PROGRAM P_AxisControl
VAR
END_VAR

//Axis Control program based on youtube series Twincat 3 NC Videos MB05a until MB17b plus MB22 by @electricalautomation https://www.youtube.com/watch?v=BxRAOdTks9I&list=PL762SfoJC-e8NbAUQ-H7a_TOdqrlBPCw4&index=25

IF G_Inputs.bManualModeSelector THEN
	Manual_mode();
ELSIF G_Inputs.bAutoModeSelector THEN
	Auto_mode();
ELSE
	GVL_AXIS1.lrBC_PowerOverride := 0;
	GVL_AXIS1.bBC_StopExe := TRUE;
	GVL_AXIS2.lrSJ_PowerOverride := 0;
	GVL_AXIS2.bSJ_StopExe := TRUE;
	GVL_AXIS3.lrTC_PowerOverride := 0;
	GVL_AXIS3.bTC_StopExe := TRUE;
	GVL_AXIS4.lrWM_PowerOverride := 0;
	GVL_AXIS4.bWM_StopExe := TRUE;
END_IF

METHOD Auto_mode : BOOL
VAR_INPUT
END_VAR
//AXIS 1 Main arm actuator

GVL_AXIS1.lrBC_PowerOverride := 100;

GVL_AXIS1.bBC_ResetExe := G_Inputs.bJoystickLeftEnable OR G_Inputs.bGreenButton OR GVL_AXIS1.bBC_MoveAbsDone;

//Power Enable
GVL_AXIS1.bBC_PowerEnCmd := G_Inputs.bAutoModeSelector;
GVL_AXIS1.bBC_PowerEnNegative := G_Inputs.bAutoModeSelector;
GVL_AXIS1.bBC_PowerEnPositive := G_Inputs.bAutoModeSelector;

GVL_AXIS1.lrBC_MoveAbsPosition := GVL_InverseKinematics.fStrokeActuatorMainInverse*1000;
GVL_AXIS1.lrBC_MoveAbsVelocity := 30;
GVL_AXIS1.bBC_MoveAbsExe := G_Inputs.bGreenButton;


//Position control
IF G_Inputs.bJoystickLeftEnable AND GVL_AXIS1.bBC_MoveAbsDone THEN
	GVL_AXIS1.bBC_ExtSetGenDisExe := FALSE;
	GVL_AXIS1.bBC_ExtSetGenEnaExe := TRUE;
ELSE
	GVL_AXIS1.bBC_ExtSetGenDisExe := TRUE;
	GVL_AXIS1.bBC_ExtSetGenEnaExe := FALSE;
END_IF


GVL_AXIS1.lrBC_MoveAddPos := GVL_InverseKinematics.fStrokeActuatorMainInverse*1000;


//Update axis
AXIS1_LD_Auto();


//Axis 3 Knuckle arm actuator

GVL_AXIS3.lrTC_PowerOverride := 100;

GVL_AXIS3.bTC_ResetExe := G_Inputs.bJoystickLeftEnable OR G_Inputs.bGreenButton OR GVL_AXIS3.bTC_MoveAbsDone;

//Power Enable
GVL_AXIS3.bTC_PowerEnCmd := G_Inputs.bAutoModeSelector;
GVL_AXIS3.bTC_PowerEnNegative := G_Inputs.bAutoModeSelector;
GVL_AXIS3.bTC_PowerEnPositive := G_Inputs.bAutoModeSelector;

GVL_AXIS3.lrTC_MoveAbsPosition := GVL_InverseKinematics.fStrokeActuatorKnuckleInverse*1000;
GVL_AXIS3.lrTC_MoveAbsVelocity := 30;
GVL_AXIS3.bTC_MoveAbsExe := G_Inputs.bGreenButton;


//Position control
IF G_Inputs.bJoystickLeftEnable AND GVL_AXIS3.bTC_MoveAbsDone THEN
	GVL_AXIS3.bTC_ExtSetGenDisExe := FALSE;
	GVL_AXIS3.bTC_ExtSetGenEnaExe := TRUE;
ELSE
	GVL_AXIS3.bTC_ExtSetGenDisExe := TRUE;
	GVL_AXIS3.bTC_ExtSetGenEnaExe := FALSE;
END_IF


GVL_AXIS3.lrTC_MoveAddPos := GVL_InverseKinematics.fStrokeActuatorKnuckleInverse*1000;


//Update axis
AXIS3_LD_Auto();


//Axis 4 Winch motor

GVL_AXIS4.lrWM_PowerOverride := 100;

GVL_AXIS4.bWM_ResetExe := G_Inputs.bJoystickRightEnable OR G_Inputs.bGreenButton OR GVL_AXIS1.bBC_MoveAbsDone;

//Power Enable
GVL_AXIS4.bWM_PowerEnCmd := G_Inputs.bAutoModeSelector;
GVL_AXIS4.bWM_PowerEnNegative := G_Inputs.bAutoModeSelector;
GVL_AXIS4.bWM_PowerEnPositive := G_Inputs.bAutoModeSelector;


GVL_AXIS4.lrWM_MoveAbsPosition := G_MachineControl.fWinchMotorAngleRef;
GVL_AXIS4.lrWM_MoveAbsVelocity := 10;
GVL_AXIS4.bWM_MoveAbsExe := G_Inputs.bGreenButton;


//Position control
IF G_Inputs.bJoystickRightEnable AND GVL_AXIS4.bWM_MoveAbsDone  THEN
	GVL_AXIS4.bWM_ExtSetGenDisExe := FALSE;
	GVL_AXIS4.bWM_ExtSetGenEnaExe := TRUE;
ELSE
	GVL_AXIS4.bWM_ExtSetGenDisExe := TRUE;
	GVL_AXIS4.bWM_ExtSetGenEnaExe := FALSE;
END_IF

(*
//Position control
IF G_Inputs.bJoystickRightEnable THEN
	GVL_AXIS4.bWM_ExtSetGenDisExe := FALSE;
	GVL_AXIS4.bWM_ExtSetGenEnaExe := TRUE;
ELSE
	GVL_AXIS4.bWM_ExtSetGenDisExe := TRUE;
	GVL_AXIS4.bWM_ExtSetGenEnaExe := FALSE;
END_IF
*)

GVL_AXIS4.lrWM_MoveAddPos := G_MachineControl.fPosRefWinch*180/PI; //Convert to degrees


//Update axis
AXIS4_LD_Auto();
END_METHOD

METHOD AXIS1_LD : BOOL
VAR_INPUT
END_VAR
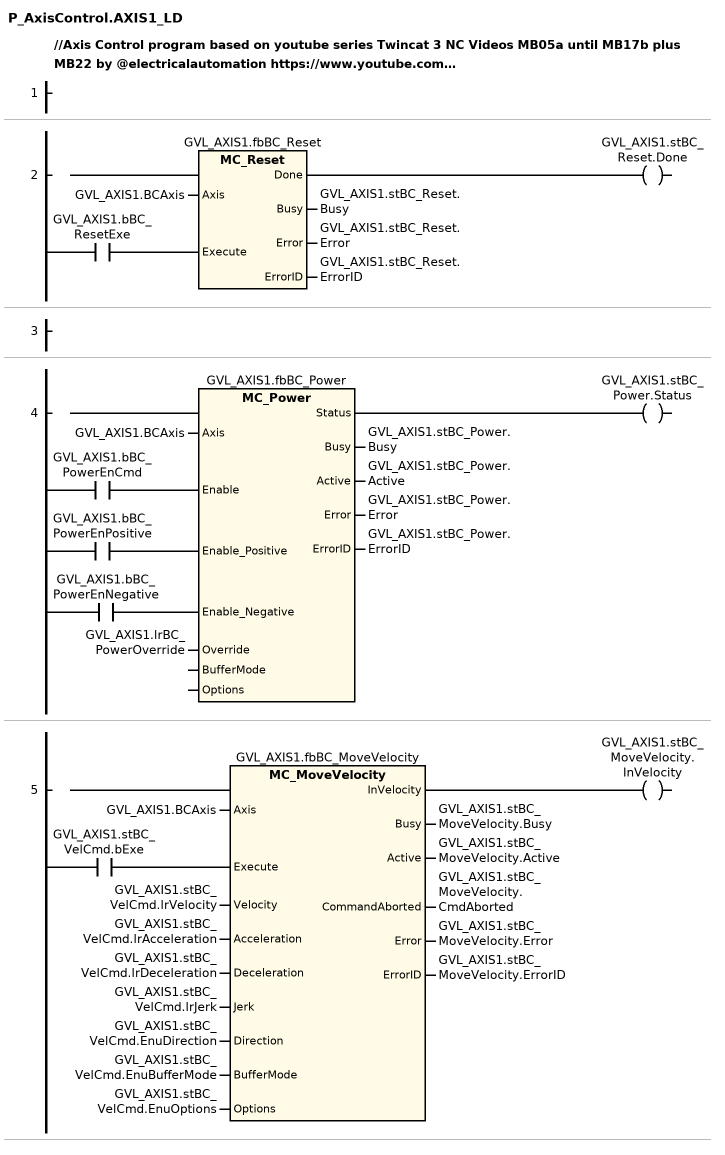
// NETWORK 1: //Axis Control program based on youtube series Twincat 3 NC Videos MB05a until MB17b plus MB22 by @electricalautomation https://www.youtube.com/watch?v=BxRAOdTks9I&list=PL762SfoJC-e8NbAUQ-H7a_TOdqrlBPCw4&index=25

// NETWORK 2
GVL_AXIS1.fbBC_Reset(
    Axis := GVL_AXIS1.BCAxis,
    Execute := GVL_AXIS1.bBC_ResetExe,
    Busy => GVL_AXIS1.stBC_Reset.Busy,
    Error => GVL_AXIS1.stBC_Reset.Error,
    ErrorID => GVL_AXIS1.stBC_Reset.ErrorID); // MC_Reset
GVL_AXIS1.stBC_Reset.Done := GVL_AXIS1.fbBC_Reset.Done;

// NETWORK 3

// NETWORK 4
GVL_AXIS1.fbBC_Power(
    Axis := GVL_AXIS1.BCAxis,
    Enable := GVL_AXIS1.bBC_PowerEnCmd,
    Enable_Positive := GVL_AXIS1.bBC_PowerEnPositive,
    Enable_Negative := GVL_AXIS1.bBC_PowerEnNegative,
    Override := GVL_AXIS1.lrBC_PowerOverride,
    Busy => GVL_AXIS1.stBC_Power.Busy,
    Active => GVL_AXIS1.stBC_Power.Active,
    Error => GVL_AXIS1.stBC_Power.Error,
    ErrorID => GVL_AXIS1.stBC_Power.ErrorID); // MC_Power
GVL_AXIS1.stBC_Power.Status := GVL_AXIS1.fbBC_Power.Status;

// NETWORK 5
GVL_AXIS1.fbBC_MoveVelocity(
    Axis := GVL_AXIS1.BCAxis,
    Execute := GVL_AXIS1.stBC_VelCmd.bExe,
    Velocity := GVL_AXIS1.stBC_VelCmd.lrVelocity,
    Acceleration := GVL_AXIS1.stBC_VelCmd.lrAcceleration,
    Deceleration := GVL_AXIS1.stBC_VelCmd.lrDeceleration,
    Jerk := GVL_AXIS1.stBC_VelCmd.lrJerk,
    Direction := GVL_AXIS1.stBC_VelCmd.EnuDirection,
    BufferMode := GVL_AXIS1.stBC_VelCmd.EnuBufferMode,
    Options := GVL_AXIS1.stBC_VelCmd.EnuOptions,
    Busy => GVL_AXIS1.stBC_MoveVelocity.Busy,
    Active => GVL_AXIS1.stBC_MoveVelocity.Active,
    CommandAborted => GVL_AXIS1.stBC_MoveVelocity.CmdAborted,
    Error => GVL_AXIS1.stBC_MoveVelocity.Error,
    ErrorID => GVL_AXIS1.stBC_MoveVelocity.ErrorID); // MC_MoveVelocity
GVL_AXIS1.stBC_MoveVelocity.InVelocity := GVL_AXIS1.fbBC_MoveVelocity.InVelocity;
END_METHOD

METHOD AXIS1_LD_Auto : BOOL
VAR_INPUT
END_VAR
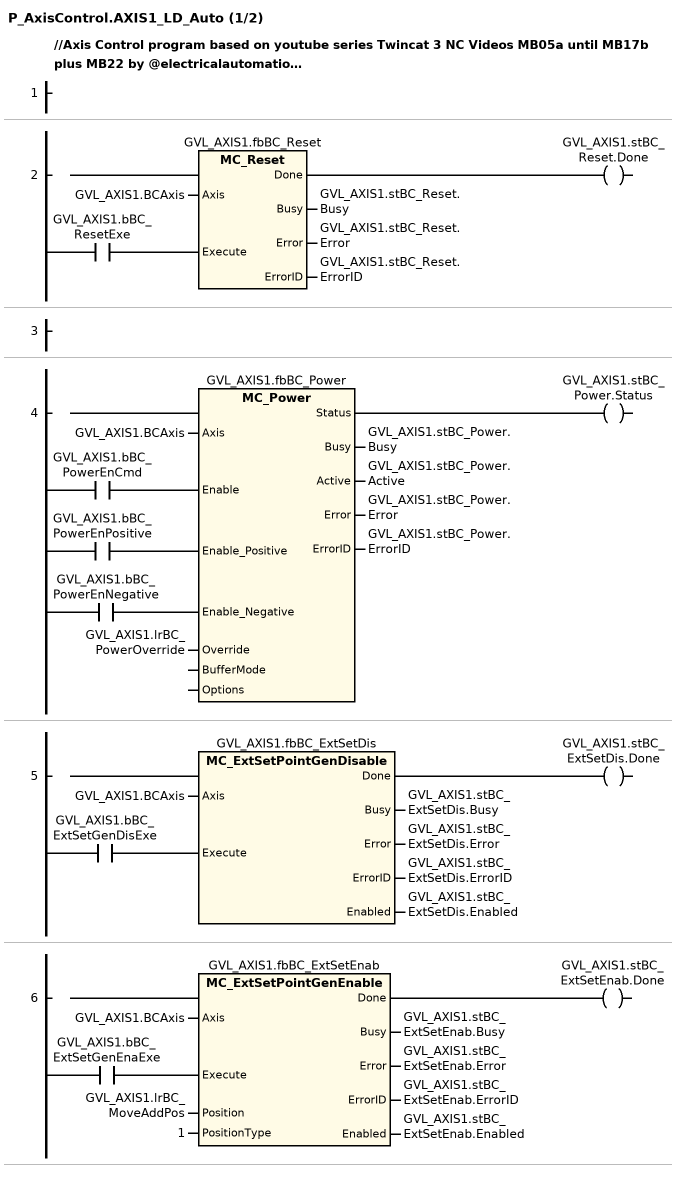
// NETWORK 1: //Axis Control program based on youtube series Twincat 3 NC Videos MB05a until MB17b plus MB22 by @electricalautomation https://www.youtube.com/watch?v=BxRAOdTks9I&list=PL762SfoJC-e8NbAUQ-H7a_TOdqrlBPCw4&index=25

// NETWORK 2
GVL_AXIS1.fbBC_Reset(
    Axis := GVL_AXIS1.BCAxis,
    Execute := GVL_AXIS1.bBC_ResetExe,
    Busy => GVL_AXIS1.stBC_Reset.Busy,
    Error => GVL_AXIS1.stBC_Reset.Error,
    ErrorID => GVL_AXIS1.stBC_Reset.ErrorID); // MC_Reset
GVL_AXIS1.stBC_Reset.Done := GVL_AXIS1.fbBC_Reset.Done;

// NETWORK 3

// NETWORK 4
GVL_AXIS1.fbBC_Power(
    Axis := GVL_AXIS1.BCAxis,
    Enable := GVL_AXIS1.bBC_PowerEnCmd,
    Enable_Positive := GVL_AXIS1.bBC_PowerEnPositive,
    Enable_Negative := GVL_AXIS1.bBC_PowerEnNegative,
    Override := GVL_AXIS1.lrBC_PowerOverride,
    Busy => GVL_AXIS1.stBC_Power.Busy,
    Active => GVL_AXIS1.stBC_Power.Active,
    Error => GVL_AXIS1.stBC_Power.Error,
    ErrorID => GVL_AXIS1.stBC_Power.ErrorID); // MC_Power
GVL_AXIS1.stBC_Power.Status := GVL_AXIS1.fbBC_Power.Status;

// NETWORK 5
GVL_AXIS1.fbBC_ExtSetDis(
    Axis := GVL_AXIS1.BCAxis,
    Execute := GVL_AXIS1.bBC_ExtSetGenDisExe,
    Busy => GVL_AXIS1.stBC_ExtSetDis.Busy,
    Error => GVL_AXIS1.stBC_ExtSetDis.Error,
    ErrorID => GVL_AXIS1.stBC_ExtSetDis.ErrorID,
    Enabled => GVL_AXIS1.stBC_ExtSetDis.Enabled); // MC_ExtSetPointGenDisable
GVL_AXIS1.stBC_ExtSetDis.Done := GVL_AXIS1.fbBC_ExtSetDis.Done;

// NETWORK 6
GVL_AXIS1.fbBC_ExtSetEnab(
    Axis := GVL_AXIS1.BCAxis,
    Execute := GVL_AXIS1.bBC_ExtSetGenEnaExe,
    Position := GVL_AXIS1.lrBC_MoveAddPos,
    PositionType := 1,
    Busy => GVL_AXIS1.stBC_ExtSetEnab.Busy,
    Error => GVL_AXIS1.stBC_ExtSetEnab.Error,
    ErrorID => GVL_AXIS1.stBC_ExtSetEnab.ErrorID,
    Enabled => GVL_AXIS1.stBC_ExtSetEnab.Enabled); // MC_ExtSetPointGenEnable
GVL_AXIS1.stBC_ExtSetEnab.Done := GVL_AXIS1.fbBC_ExtSetEnab.Done;

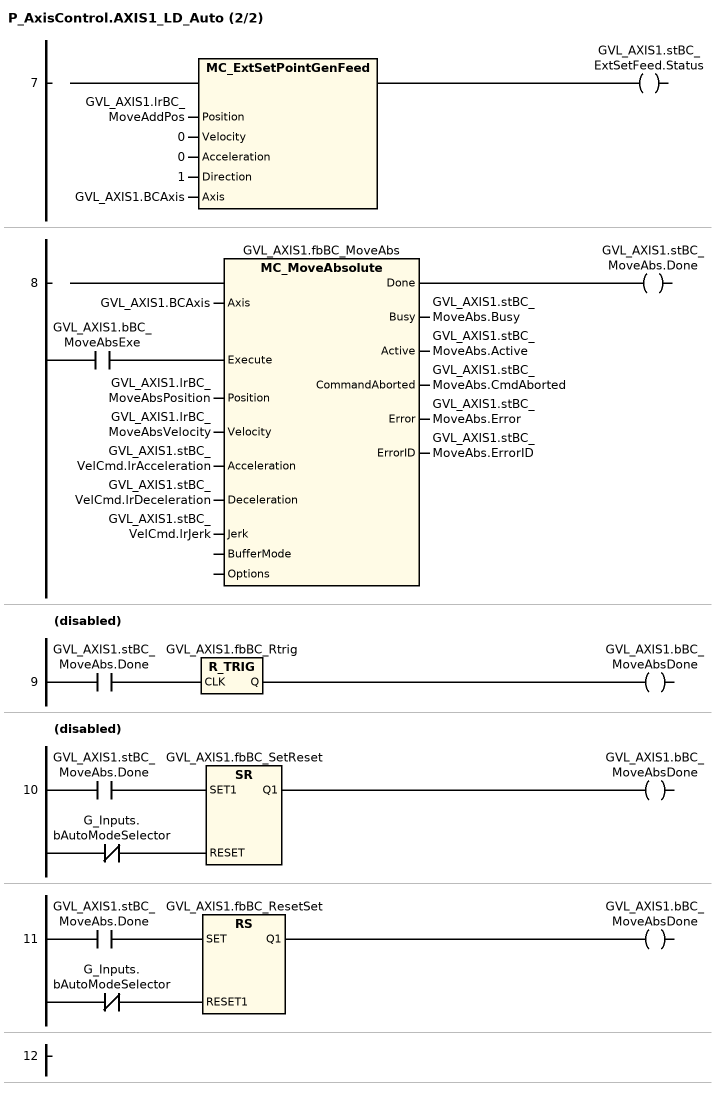
// NETWORK 7
GVL_AXIS1.stBC_ExtSetFeed.Status := MC_ExtSetPointGenFeed(Position := GVL_AXIS1.lrBC_MoveAddPos, Velocity := 0, Acceleration := 0, Direction := 1, Axis := GVL_AXIS1.BCAxis);

// NETWORK 8
GVL_AXIS1.fbBC_MoveAbs(
    Axis := GVL_AXIS1.BCAxis,
    Execute := GVL_AXIS1.bBC_MoveAbsExe,
    Position := GVL_AXIS1.lrBC_MoveAbsPosition,
    Velocity := GVL_AXIS1.lrBC_MoveAbsVelocity,
    Acceleration := GVL_AXIS1.stBC_VelCmd.lrAcceleration,
    Deceleration := GVL_AXIS1.stBC_VelCmd.lrDeceleration,
    Jerk := GVL_AXIS1.stBC_VelCmd.lrJerk,
    Busy => GVL_AXIS1.stBC_MoveAbs.Busy,
    Active => GVL_AXIS1.stBC_MoveAbs.Active,
    CommandAborted => GVL_AXIS1.stBC_MoveAbs.CmdAborted,
    Error => GVL_AXIS1.stBC_MoveAbs.Error,
    ErrorID => GVL_AXIS1.stBC_MoveAbs.ErrorID); // MC_MoveAbsolute
GVL_AXIS1.stBC_MoveAbs.Done := GVL_AXIS1.fbBC_MoveAbs.Done;

// NETWORK 9 (disabled)
// GVL_AXIS1.fbBC_Rtrig(CLK := GVL_AXIS1.stBC_MoveAbs.Done); // R_TRIG
// GVL_AXIS1.bBC_MoveAbsDone := GVL_AXIS1.fbBC_Rtrig.Q;

// NETWORK 10 (disabled)
// GVL_AXIS1.fbBC_SetReset(SET1 := GVL_AXIS1.stBC_MoveAbs.Done, RESET := NOT G_Inputs.bAutoModeSelector); // SR
// GVL_AXIS1.bBC_MoveAbsDone := GVL_AXIS1.fbBC_SetReset.Q1;

// NETWORK 11
GVL_AXIS1.fbBC_ResetSet(SET := GVL_AXIS1.stBC_MoveAbs.Done, RESET1 := NOT G_Inputs.bAutoModeSelector); // RS
GVL_AXIS1.bBC_MoveAbsDone := GVL_AXIS1.fbBC_ResetSet.Q1;

// NETWORK 12
END_METHOD

METHOD AXIS2_LD : BOOL
VAR_INPUT
END_VAR
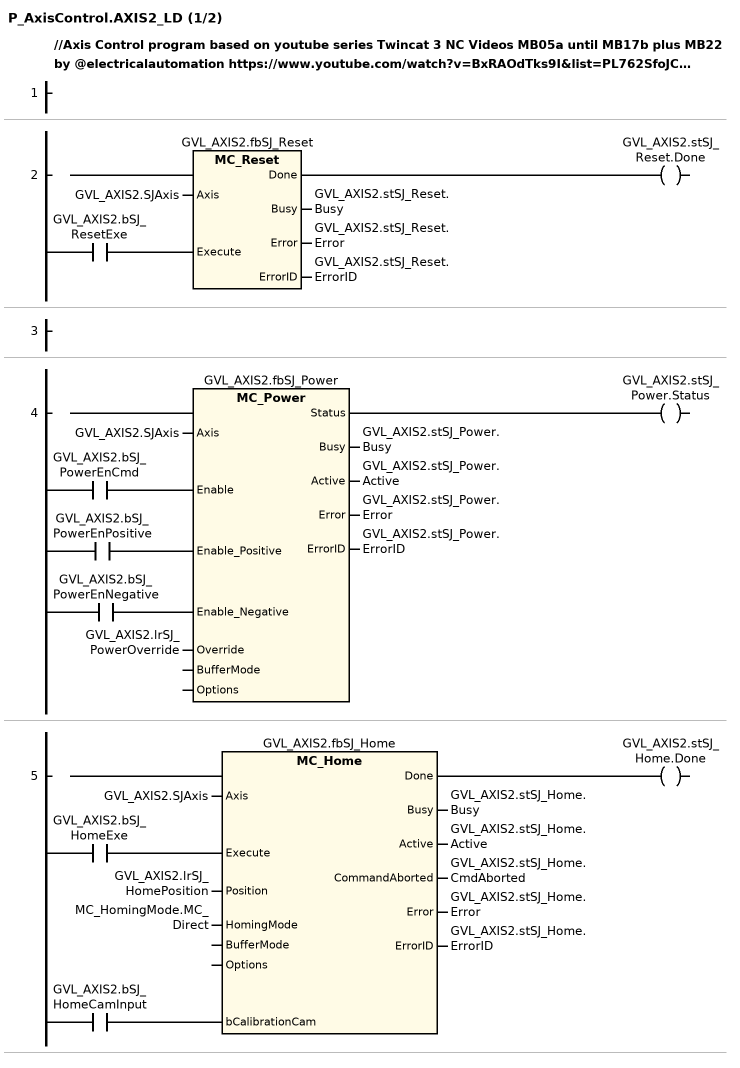
// NETWORK 1: //Axis Control program based on youtube series Twincat 3 NC Videos MB05a until MB17b plus MB22 by @electricalautomation https://www.youtube.com/watch?v=BxRAOdTks9I&list=PL762SfoJC-e8NbAUQ-H7a_TOdqrlBPCw4&index=25

// NETWORK 2
GVL_AXIS2.fbSJ_Reset(
    Axis := GVL_AXIS2.SJAxis,
    Execute := GVL_AXIS2.bSJ_ResetExe,
    Busy => GVL_AXIS2.stSJ_Reset.Busy,
    Error => GVL_AXIS2.stSJ_Reset.Error,
    ErrorID => GVL_AXIS2.stSJ_Reset.ErrorID); // MC_Reset
GVL_AXIS2.stSJ_Reset.Done := GVL_AXIS2.fbSJ_Reset.Done;

// NETWORK 3

// NETWORK 4
GVL_AXIS2.fbSJ_Power(
    Axis := GVL_AXIS2.SJAxis,
    Enable := GVL_AXIS2.bSJ_PowerEnCmd,
    Enable_Positive := GVL_AXIS2.bSJ_PowerEnPositive,
    Enable_Negative := GVL_AXIS2.bSJ_PowerEnNegative,
    Override := GVL_AXIS2.lrSJ_PowerOverride,
    Busy => GVL_AXIS2.stSJ_Power.Busy,
    Active => GVL_AXIS2.stSJ_Power.Active,
    Error => GVL_AXIS2.stSJ_Power.Error,
    ErrorID => GVL_AXIS2.stSJ_Power.ErrorID); // MC_Power
GVL_AXIS2.stSJ_Power.Status := GVL_AXIS2.fbSJ_Power.Status;

// NETWORK 5
GVL_AXIS2.fbSJ_Home(
    Axis := GVL_AXIS2.SJAxis,
    Execute := GVL_AXIS2.bSJ_HomeExe,
    Position := GVL_AXIS2.lrSJ_HomePosition,
    HomingMode := MC_HomingMode.MC_Direct,
    bCalibrationCam := GVL_AXIS2.bSJ_HomeCamInput,
    Busy => GVL_AXIS2.stSJ_Home.Busy,
    Active => GVL_AXIS2.stSJ_Home.Active,
    CommandAborted => GVL_AXIS2.stSJ_Home.CmdAborted,
    Error => GVL_AXIS2.stSJ_Home.Error,
    ErrorID => GVL_AXIS2.stSJ_Home.ErrorID); // MC_Home
GVL_AXIS2.stSJ_Home.Done := GVL_AXIS2.fbSJ_Home.Done;

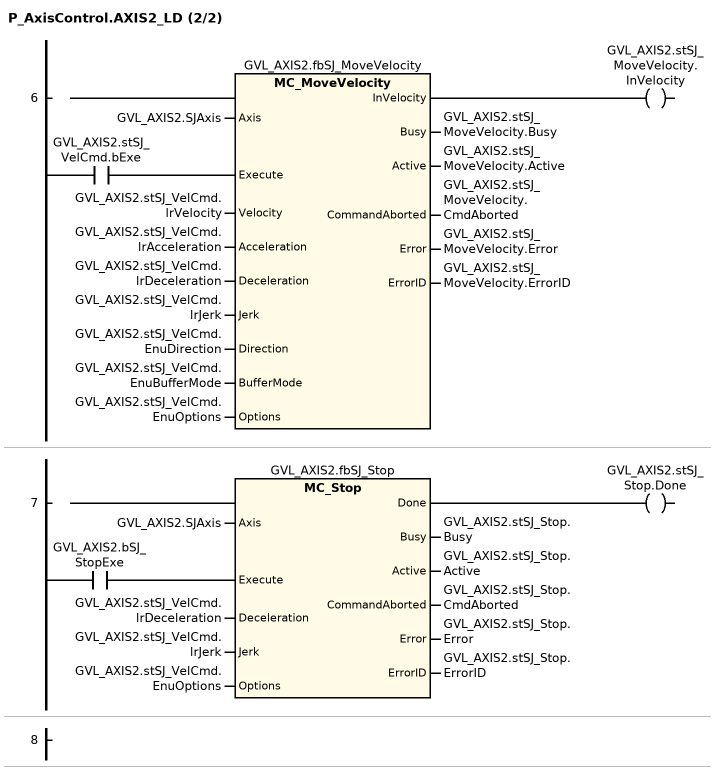
// NETWORK 6
GVL_AXIS2.fbSJ_MoveVelocity(
    Axis := GVL_AXIS2.SJAxis,
    Execute := GVL_AXIS2.stSJ_VelCmd.bExe,
    Velocity := GVL_AXIS2.stSJ_VelCmd.lrVelocity,
    Acceleration := GVL_AXIS2.stSJ_VelCmd.lrAcceleration,
    Deceleration := GVL_AXIS2.stSJ_VelCmd.lrDeceleration,
    Jerk := GVL_AXIS2.stSJ_VelCmd.lrJerk,
    Direction := GVL_AXIS2.stSJ_VelCmd.EnuDirection,
    BufferMode := GVL_AXIS2.stSJ_VelCmd.EnuBufferMode,
    Options := GVL_AXIS2.stSJ_VelCmd.EnuOptions,
    Busy => GVL_AXIS2.stSJ_MoveVelocity.Busy,
    Active => GVL_AXIS2.stSJ_MoveVelocity.Active,
    CommandAborted => GVL_AXIS2.stSJ_MoveVelocity.CmdAborted,
    Error => GVL_AXIS2.stSJ_MoveVelocity.Error,
    ErrorID => GVL_AXIS2.stSJ_MoveVelocity.ErrorID); // MC_MoveVelocity
GVL_AXIS2.stSJ_MoveVelocity.InVelocity := GVL_AXIS2.fbSJ_MoveVelocity.InVelocity;

// NETWORK 7
GVL_AXIS2.fbSJ_Stop(
    Axis := GVL_AXIS2.SJAxis,
    Execute := GVL_AXIS2.bSJ_StopExe,
    Deceleration := GVL_AXIS2.stSJ_VelCmd.lrDeceleration,
    Jerk := GVL_AXIS2.stSJ_VelCmd.lrJerk,
    Options := GVL_AXIS2.stSJ_VelCmd.EnuOptions,
    Busy => GVL_AXIS2.stSJ_Stop.Busy,
    Active => GVL_AXIS2.stSJ_Stop.Active,
    CommandAborted => GVL_AXIS2.stSJ_Stop.CmdAborted,
    Error => GVL_AXIS2.stSJ_Stop.Error,
    ErrorID => GVL_AXIS2.stSJ_Stop.ErrorID); // MC_Stop
GVL_AXIS2.stSJ_Stop.Done := GVL_AXIS2.fbSJ_Stop.Done;

// NETWORK 8
END_METHOD

METHOD AXIS3_LD : BOOL
VAR_INPUT
END_VAR
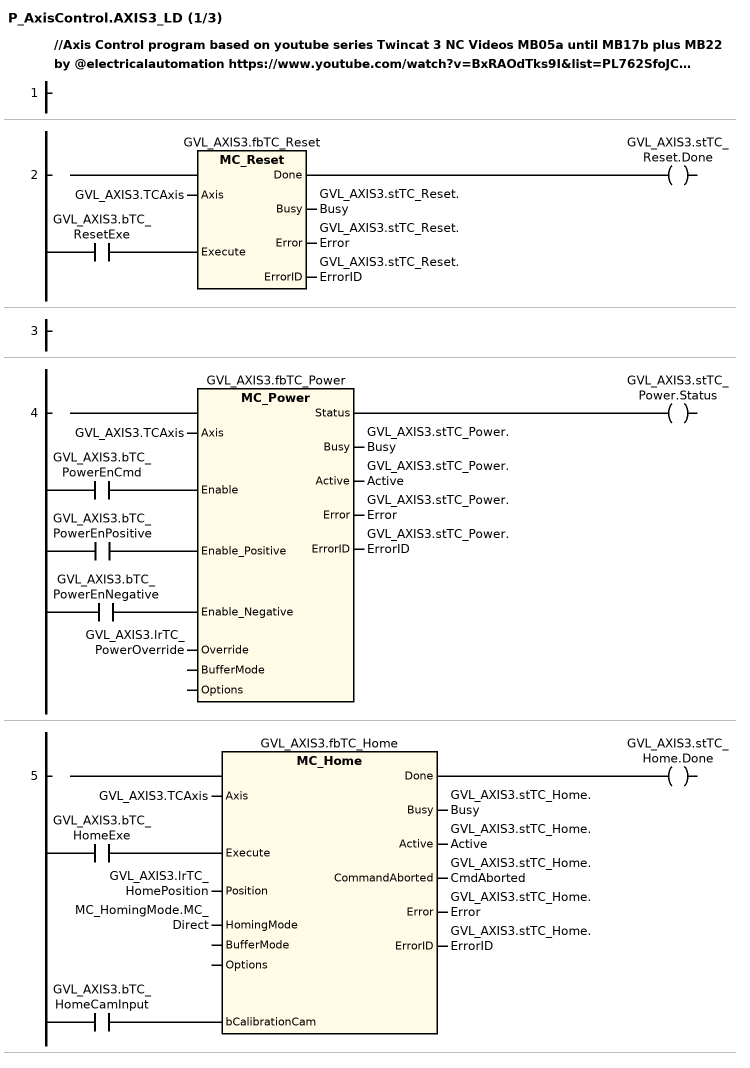
// NETWORK 1: //Axis Control program based on youtube series Twincat 3 NC Videos MB05a until MB17b plus MB22 by @electricalautomation https://www.youtube.com/watch?v=BxRAOdTks9I&list=PL762SfoJC-e8NbAUQ-H7a_TOdqrlBPCw4&index=25

// NETWORK 2
GVL_AXIS3.fbTC_Reset(
    Axis := GVL_AXIS3.TCAxis,
    Execute := GVL_AXIS3.bTC_ResetExe,
    Busy => GVL_AXIS3.stTC_Reset.Busy,
    Error => GVL_AXIS3.stTC_Reset.Error,
    ErrorID => GVL_AXIS3.stTC_Reset.ErrorID); // MC_Reset
GVL_AXIS3.stTC_Reset.Done := GVL_AXIS3.fbTC_Reset.Done;

// NETWORK 3

// NETWORK 4
GVL_AXIS3.fbTC_Power(
    Axis := GVL_AXIS3.TCAxis,
    Enable := GVL_AXIS3.bTC_PowerEnCmd,
    Enable_Positive := GVL_AXIS3.bTC_PowerEnPositive,
    Enable_Negative := GVL_AXIS3.bTC_PowerEnNegative,
    Override := GVL_AXIS3.lrTC_PowerOverride,
    Busy => GVL_AXIS3.stTC_Power.Busy,
    Active => GVL_AXIS3.stTC_Power.Active,
    Error => GVL_AXIS3.stTC_Power.Error,
    ErrorID => GVL_AXIS3.stTC_Power.ErrorID); // MC_Power
GVL_AXIS3.stTC_Power.Status := GVL_AXIS3.fbTC_Power.Status;

// NETWORK 5
GVL_AXIS3.fbTC_Home(
    Axis := GVL_AXIS3.TCAxis,
    Execute := GVL_AXIS3.bTC_HomeExe,
    Position := GVL_AXIS3.lrTC_HomePosition,
    HomingMode := MC_HomingMode.MC_Direct,
    bCalibrationCam := GVL_AXIS3.bTC_HomeCamInput,
    Busy => GVL_AXIS3.stTC_Home.Busy,
    Active => GVL_AXIS3.stTC_Home.Active,
    CommandAborted => GVL_AXIS3.stTC_Home.CmdAborted,
    Error => GVL_AXIS3.stTC_Home.Error,
    ErrorID => GVL_AXIS3.stTC_Home.ErrorID); // MC_Home
GVL_AXIS3.stTC_Home.Done := GVL_AXIS3.fbTC_Home.Done;

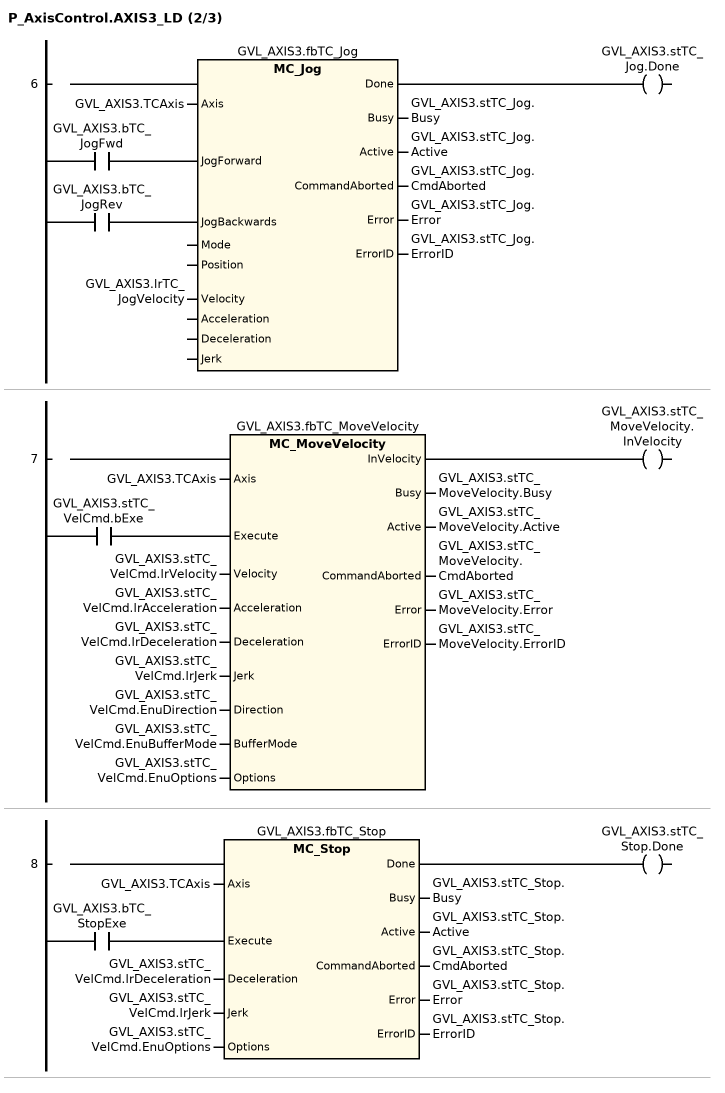
// NETWORK 6
GVL_AXIS3.fbTC_Jog(
    Axis := GVL_AXIS3.TCAxis,
    JogForward := GVL_AXIS3.bTC_JogFwd,
    JogBackwards := GVL_AXIS3.bTC_JogRev,
    Velocity := GVL_AXIS3.lrTC_JogVelocity,
    Busy => GVL_AXIS3.stTC_Jog.Busy,
    Active => GVL_AXIS3.stTC_Jog.Active,
    CommandAborted => GVL_AXIS3.stTC_Jog.CmdAborted,
    Error => GVL_AXIS3.stTC_Jog.Error,
    ErrorID => GVL_AXIS3.stTC_Jog.ErrorID); // MC_Jog
GVL_AXIS3.stTC_Jog.Done := GVL_AXIS3.fbTC_Jog.Done;

// NETWORK 7
GVL_AXIS3.fbTC_MoveVelocity(
    Axis := GVL_AXIS3.TCAxis,
    Execute := GVL_AXIS3.stTC_VelCmd.bExe,
    Velocity := GVL_AXIS3.stTC_VelCmd.lrVelocity,
    Acceleration := GVL_AXIS3.stTC_VelCmd.lrAcceleration,
    Deceleration := GVL_AXIS3.stTC_VelCmd.lrDeceleration,
    Jerk := GVL_AXIS3.stTC_VelCmd.lrJerk,
    Direction := GVL_AXIS3.stTC_VelCmd.EnuDirection,
    BufferMode := GVL_AXIS3.stTC_VelCmd.EnuBufferMode,
    Options := GVL_AXIS3.stTC_VelCmd.EnuOptions,
    Busy => GVL_AXIS3.stTC_MoveVelocity.Busy,
    Active => GVL_AXIS3.stTC_MoveVelocity.Active,
    CommandAborted => GVL_AXIS3.stTC_MoveVelocity.CmdAborted,
    Error => GVL_AXIS3.stTC_MoveVelocity.Error,
    ErrorID => GVL_AXIS3.stTC_MoveVelocity.ErrorID); // MC_MoveVelocity
GVL_AXIS3.stTC_MoveVelocity.InVelocity := GVL_AXIS3.fbTC_MoveVelocity.InVelocity;

// NETWORK 8
GVL_AXIS3.fbTC_Stop(
    Axis := GVL_AXIS3.TCAxis,
    Execute := GVL_AXIS3.bTC_StopExe,
    Deceleration := GVL_AXIS3.stTC_VelCmd.lrDeceleration,
    Jerk := GVL_AXIS3.stTC_VelCmd.lrJerk,
    Options := GVL_AXIS3.stTC_VelCmd.EnuOptions,
    Busy => GVL_AXIS3.stTC_Stop.Busy,
    Active => GVL_AXIS3.stTC_Stop.Active,
    CommandAborted => GVL_AXIS3.stTC_Stop.CmdAborted,
    Error => GVL_AXIS3.stTC_Stop.Error,
    ErrorID => GVL_AXIS3.stTC_Stop.ErrorID); // MC_Stop
GVL_AXIS3.stTC_Stop.Done := GVL_AXIS3.fbTC_Stop.Done;

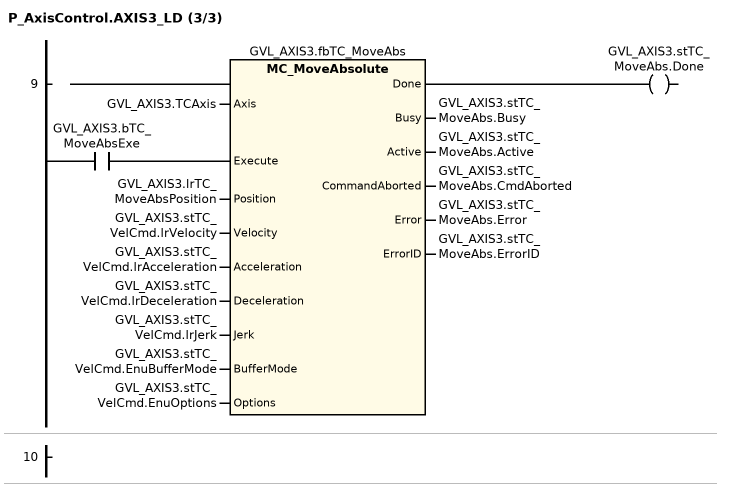
// NETWORK 9
GVL_AXIS3.fbTC_MoveAbs(
    Axis := GVL_AXIS3.TCAxis,
    Execute := GVL_AXIS3.bTC_MoveAbsExe,
    Position := GVL_AXIS3.lrTC_MoveAbsPosition,
    Velocity := GVL_AXIS3.stTC_VelCmd.lrVelocity,
    Acceleration := GVL_AXIS3.stTC_VelCmd.lrAcceleration,
    Deceleration := GVL_AXIS3.stTC_VelCmd.lrDeceleration,
    Jerk := GVL_AXIS3.stTC_VelCmd.lrJerk,
    BufferMode := GVL_AXIS3.stTC_VelCmd.EnuBufferMode,
    Options := GVL_AXIS3.stTC_VelCmd.EnuOptions,
    Busy => GVL_AXIS3.stTC_MoveAbs.Busy,
    Active => GVL_AXIS3.stTC_MoveAbs.Active,
    CommandAborted => GVL_AXIS3.stTC_MoveAbs.CmdAborted,
    Error => GVL_AXIS3.stTC_MoveAbs.Error,
    ErrorID => GVL_AXIS3.stTC_MoveAbs.ErrorID); // MC_MoveAbsolute
GVL_AXIS3.stTC_MoveAbs.Done := GVL_AXIS3.fbTC_MoveAbs.Done;

// NETWORK 10
END_METHOD

METHOD AXIS3_LD_Auto : BOOL
VAR_INPUT
END_VAR
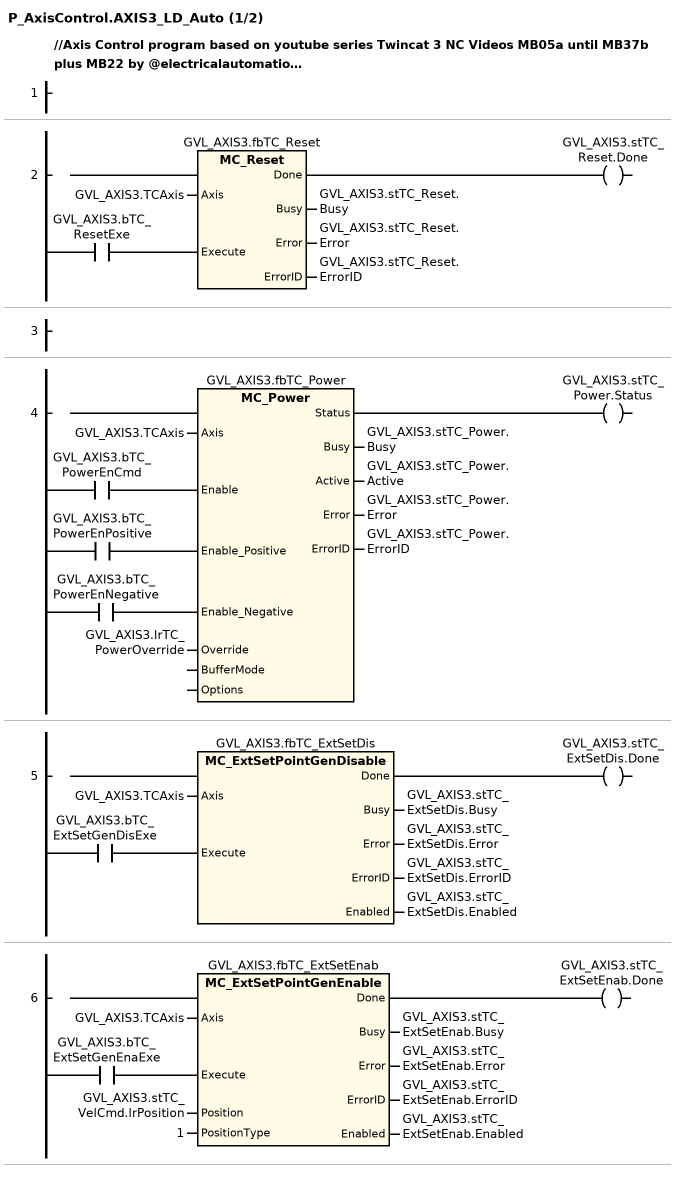
// NETWORK 1: //Axis Control program based on youtube series Twincat 3 NC Videos MB05a until MB37b plus MB22 by @electricalautomation https://www.youtube.com/watch?v=BxRAOdTks9I&list=PL762SfoJC-e8NbAUQ-H7a_TOdqrlBPCw4&index=25

// NETWORK 2
GVL_AXIS3.fbTC_Reset(
    Axis := GVL_AXIS3.TCAxis,
    Execute := GVL_AXIS3.bTC_ResetExe,
    Busy => GVL_AXIS3.stTC_Reset.Busy,
    Error => GVL_AXIS3.stTC_Reset.Error,
    ErrorID => GVL_AXIS3.stTC_Reset.ErrorID); // MC_Reset
GVL_AXIS3.stTC_Reset.Done := GVL_AXIS3.fbTC_Reset.Done;

// NETWORK 3

// NETWORK 4
GVL_AXIS3.fbTC_Power(
    Axis := GVL_AXIS3.TCAxis,
    Enable := GVL_AXIS3.bTC_PowerEnCmd,
    Enable_Positive := GVL_AXIS3.bTC_PowerEnPositive,
    Enable_Negative := GVL_AXIS3.bTC_PowerEnNegative,
    Override := GVL_AXIS3.lrTC_PowerOverride,
    Busy => GVL_AXIS3.stTC_Power.Busy,
    Active => GVL_AXIS3.stTC_Power.Active,
    Error => GVL_AXIS3.stTC_Power.Error,
    ErrorID => GVL_AXIS3.stTC_Power.ErrorID); // MC_Power
GVL_AXIS3.stTC_Power.Status := GVL_AXIS3.fbTC_Power.Status;

// NETWORK 5
GVL_AXIS3.fbTC_ExtSetDis(
    Axis := GVL_AXIS3.TCAxis,
    Execute := GVL_AXIS3.bTC_ExtSetGenDisExe,
    Busy => GVL_AXIS3.stTC_ExtSetDis.Busy,
    Error => GVL_AXIS3.stTC_ExtSetDis.Error,
    ErrorID => GVL_AXIS3.stTC_ExtSetDis.ErrorID,
    Enabled => GVL_AXIS3.stTC_ExtSetDis.Enabled); // MC_ExtSetPointGenDisable
GVL_AXIS3.stTC_ExtSetDis.Done := GVL_AXIS3.fbTC_ExtSetDis.Done;

// NETWORK 6
GVL_AXIS3.fbTC_ExtSetEnab(
    Axis := GVL_AXIS3.TCAxis,
    Execute := GVL_AXIS3.bTC_ExtSetGenEnaExe,
    Position := GVL_AXIS3.stTC_VelCmd.lrPosition,
    PositionType := 1,
    Busy => GVL_AXIS3.stTC_ExtSetEnab.Busy,
    Error => GVL_AXIS3.stTC_ExtSetEnab.Error,
    ErrorID => GVL_AXIS3.stTC_ExtSetEnab.ErrorID,
    Enabled => GVL_AXIS3.stTC_ExtSetEnab.Enabled); // MC_ExtSetPointGenEnable
GVL_AXIS3.stTC_ExtSetEnab.Done := GVL_AXIS3.fbTC_ExtSetEnab.Done;

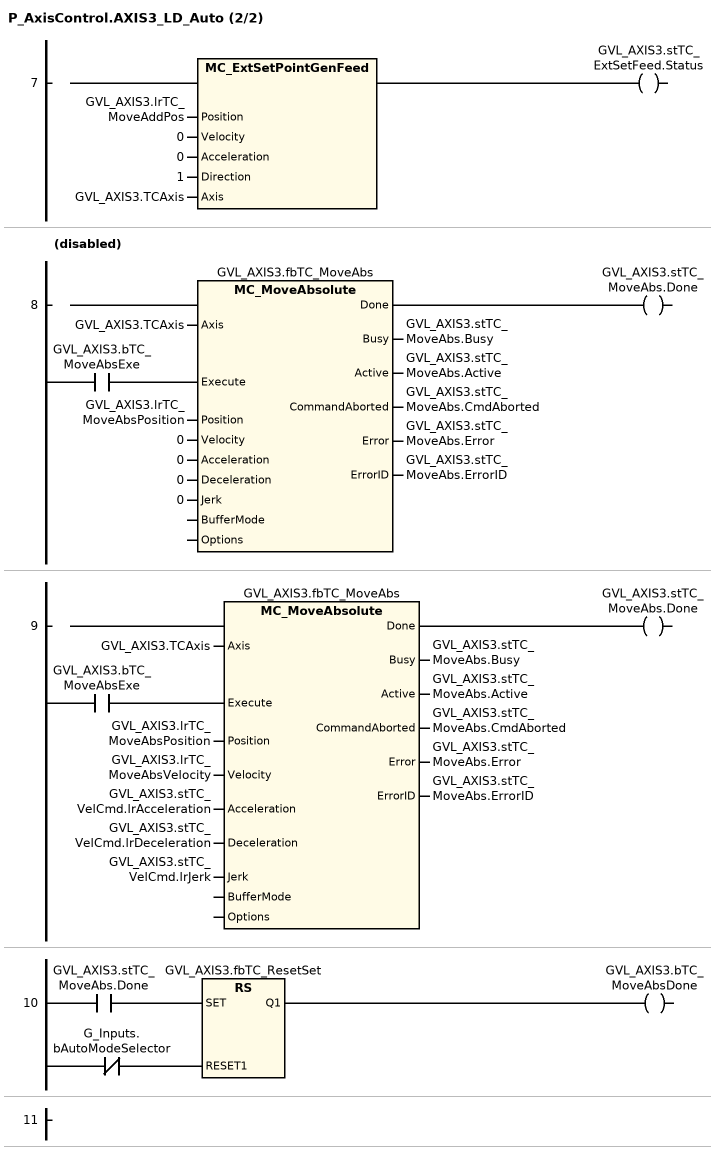
// NETWORK 7
GVL_AXIS3.stTC_ExtSetFeed.Status := MC_ExtSetPointGenFeed(Position := GVL_AXIS3.lrTC_MoveAddPos, Velocity := 0, Acceleration := 0, Direction := 1, Axis := GVL_AXIS3.TCAxis);

// NETWORK 8 (disabled)
// GVL_AXIS3.fbTC_MoveAbs(
//     Axis := GVL_AXIS3.TCAxis,
//     Execute := GVL_AXIS3.bTC_MoveAbsExe,
//     Position := GVL_AXIS3.lrTC_MoveAbsPosition,
//     Velocity := 0,
//     Acceleration := 0,
//     Deceleration := 0,
//     Jerk := 0,
//     Busy => GVL_AXIS3.stTC_MoveAbs.Busy,
//     Active => GVL_AXIS3.stTC_MoveAbs.Active,
//     CommandAborted => GVL_AXIS3.stTC_MoveAbs.CmdAborted,
//     Error => GVL_AXIS3.stTC_MoveAbs.Error,
//     ErrorID => GVL_AXIS3.stTC_MoveAbs.ErrorID); // MC_MoveAbsolute
// GVL_AXIS3.stTC_MoveAbs.Done := GVL_AXIS3.fbTC_MoveAbs.Done;

// NETWORK 9
GVL_AXIS3.fbTC_MoveAbs(
    Axis := GVL_AXIS3.TCAxis,
    Execute := GVL_AXIS3.bTC_MoveAbsExe,
    Position := GVL_AXIS3.lrTC_MoveAbsPosition,
    Velocity := GVL_AXIS3.lrTC_MoveAbsVelocity,
    Acceleration := GVL_AXIS3.stTC_VelCmd.lrAcceleration,
    Deceleration := GVL_AXIS3.stTC_VelCmd.lrDeceleration,
    Jerk := GVL_AXIS3.stTC_VelCmd.lrJerk,
    Busy => GVL_AXIS3.stTC_MoveAbs.Busy,
    Active => GVL_AXIS3.stTC_MoveAbs.Active,
    CommandAborted => GVL_AXIS3.stTC_MoveAbs.CmdAborted,
    Error => GVL_AXIS3.stTC_MoveAbs.Error,
    ErrorID => GVL_AXIS3.stTC_MoveAbs.ErrorID); // MC_MoveAbsolute
GVL_AXIS3.stTC_MoveAbs.Done := GVL_AXIS3.fbTC_MoveAbs.Done;

// NETWORK 10
GVL_AXIS3.fbTC_ResetSet(SET := GVL_AXIS3.stTC_MoveAbs.Done, RESET1 := NOT G_Inputs.bAutoModeSelector); // RS
GVL_AXIS3.bTC_MoveAbsDone := GVL_AXIS3.fbTC_ResetSet.Q1;

// NETWORK 11
END_METHOD

METHOD AXIS4_LD : BOOL
VAR_INPUT
END_VAR
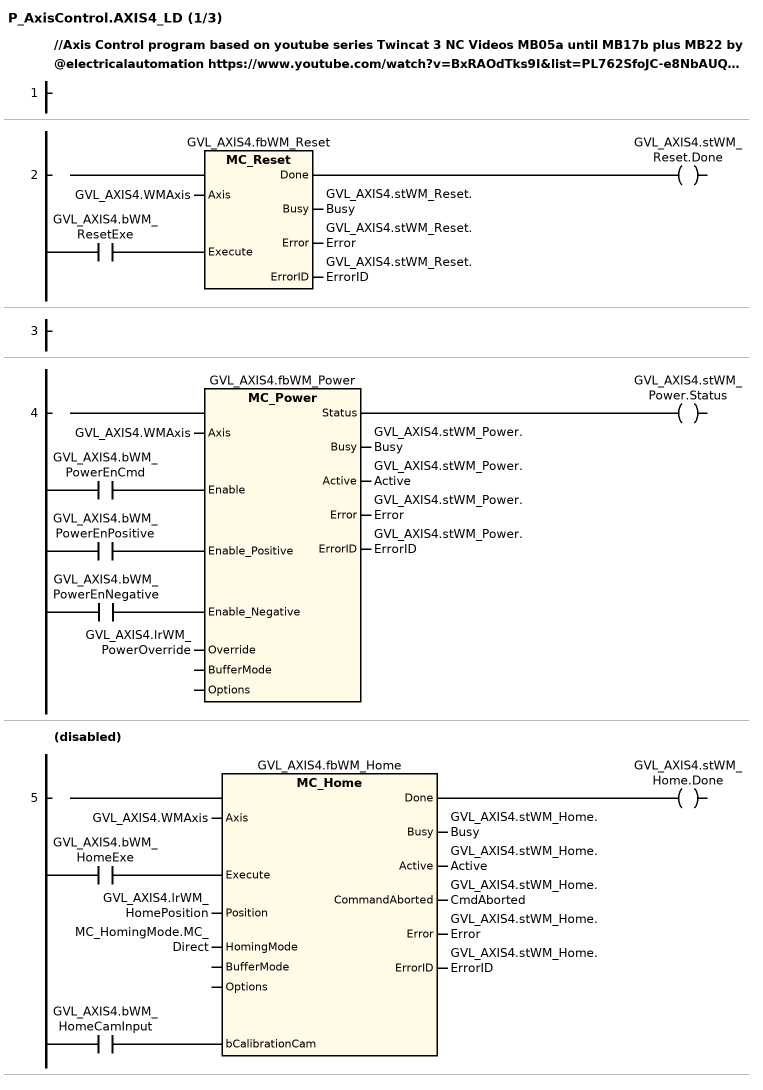
// NETWORK 1: //Axis Control program based on youtube series Twincat 3 NC Videos MB05a until MB17b plus MB22 by @electricalautomation https://www.youtube.com/watch?v=BxRAOdTks9I&list=PL762SfoJC-e8NbAUQ-H7a_TOdqrlBPCw4&index=25

// NETWORK 2
GVL_AXIS4.fbWM_Reset(
    Axis := GVL_AXIS4.WMAxis,
    Execute := GVL_AXIS4.bWM_ResetExe,
    Busy => GVL_AXIS4.stWM_Reset.Busy,
    Error => GVL_AXIS4.stWM_Reset.Error,
    ErrorID => GVL_AXIS4.stWM_Reset.ErrorID); // MC_Reset
GVL_AXIS4.stWM_Reset.Done := GVL_AXIS4.fbWM_Reset.Done;

// NETWORK 3

// NETWORK 4
GVL_AXIS4.fbWM_Power(
    Axis := GVL_AXIS4.WMAxis,
    Enable := GVL_AXIS4.bWM_PowerEnCmd,
    Enable_Positive := GVL_AXIS4.bWM_PowerEnPositive,
    Enable_Negative := GVL_AXIS4.bWM_PowerEnNegative,
    Override := GVL_AXIS4.lrWM_PowerOverride,
    Busy => GVL_AXIS4.stWM_Power.Busy,
    Active => GVL_AXIS4.stWM_Power.Active,
    Error => GVL_AXIS4.stWM_Power.Error,
    ErrorID => GVL_AXIS4.stWM_Power.ErrorID); // MC_Power
GVL_AXIS4.stWM_Power.Status := GVL_AXIS4.fbWM_Power.Status;

// NETWORK 5 (disabled)
// GVL_AXIS4.fbWM_Home(
//     Axis := GVL_AXIS4.WMAxis,
//     Execute := GVL_AXIS4.bWM_HomeExe,
//     Position := GVL_AXIS4.lrWM_HomePosition,
//     HomingMode := MC_HomingMode.MC_Direct,
//     bCalibrationCam := GVL_AXIS4.bWM_HomeCamInput,
//     Busy => GVL_AXIS4.stWM_Home.Busy,
//     Active => GVL_AXIS4.stWM_Home.Active,
//     CommandAborted => GVL_AXIS4.stWM_Home.CmdAborted,
//     Error => GVL_AXIS4.stWM_Home.Error,
//     ErrorID => GVL_AXIS4.stWM_Home.ErrorID); // MC_Home
// GVL_AXIS4.stWM_Home.Done := GVL_AXIS4.fbWM_Home.Done;

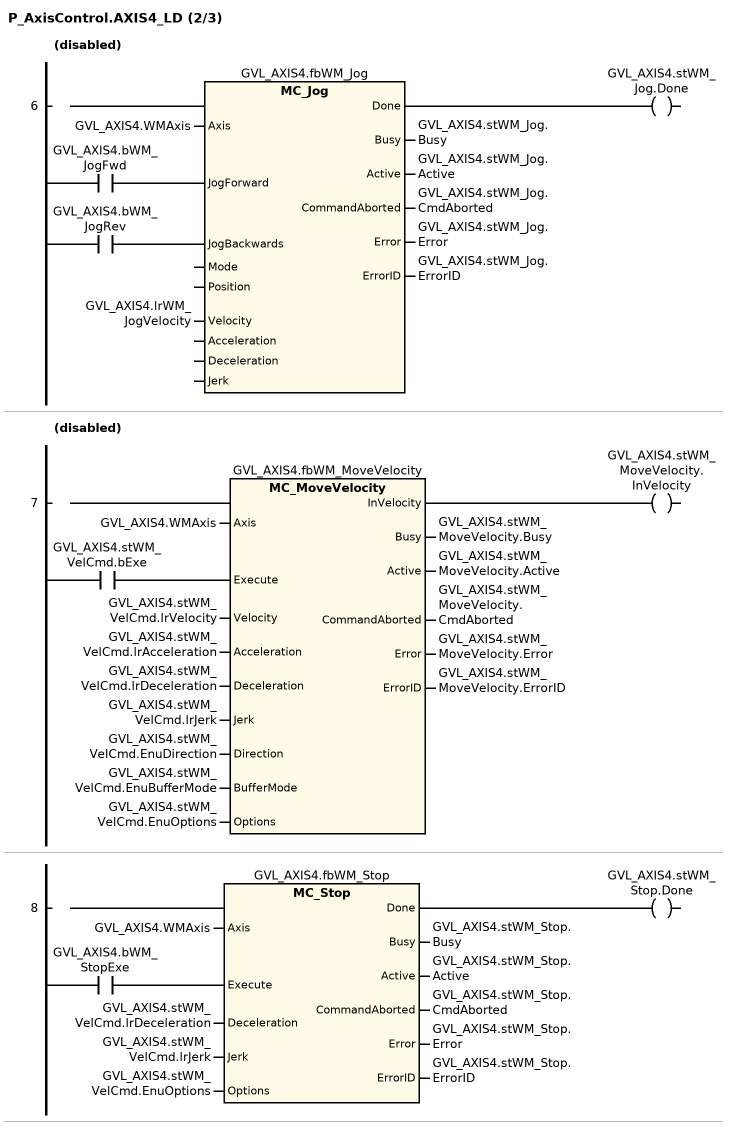
// NETWORK 6 (disabled)
// GVL_AXIS4.fbWM_Jog(
//     Axis := GVL_AXIS4.WMAxis,
//     JogForward := GVL_AXIS4.bWM_JogFwd,
//     JogBackwards := GVL_AXIS4.bWM_JogRev,
//     Velocity := GVL_AXIS4.lrWM_JogVelocity,
//     Busy => GVL_AXIS4.stWM_Jog.Busy,
//     Active => GVL_AXIS4.stWM_Jog.Active,
//     CommandAborted => GVL_AXIS4.stWM_Jog.CmdAborted,
//     Error => GVL_AXIS4.stWM_Jog.Error,
//     ErrorID => GVL_AXIS4.stWM_Jog.ErrorID); // MC_Jog
// GVL_AXIS4.stWM_Jog.Done := GVL_AXIS4.fbWM_Jog.Done;

// NETWORK 7 (disabled)
// GVL_AXIS4.fbWM_MoveVelocity(
//     Axis := GVL_AXIS4.WMAxis,
//     Execute := GVL_AXIS4.stWM_VelCmd.bExe,
//     Velocity := GVL_AXIS4.stWM_VelCmd.lrVelocity,
//     Acceleration := GVL_AXIS4.stWM_VelCmd.lrAcceleration,
//     Deceleration := GVL_AXIS4.stWM_VelCmd.lrDeceleration,
//     Jerk := GVL_AXIS4.stWM_VelCmd.lrJerk,
//     Direction := GVL_AXIS4.stWM_VelCmd.EnuDirection,
//     BufferMode := GVL_AXIS4.stWM_VelCmd.EnuBufferMode,
//     Options := GVL_AXIS4.stWM_VelCmd.EnuOptions,
//     Busy => GVL_AXIS4.stWM_MoveVelocity.Busy,
//     Active => GVL_AXIS4.stWM_MoveVelocity.Active,
//     CommandAborted => GVL_AXIS4.stWM_MoveVelocity.CmdAborted,
//     Error => GVL_AXIS4.stWM_MoveVelocity.Error,
//     ErrorID => GVL_AXIS4.stWM_MoveVelocity.ErrorID); // MC_MoveVelocity
// GVL_AXIS4.stWM_MoveVelocity.InVelocity := GVL_AXIS4.fbWM_MoveVelocity.InVelocity;

// NETWORK 8
GVL_AXIS4.fbWM_Stop(
    Axis := GVL_AXIS4.WMAxis,
    Execute := GVL_AXIS4.bWM_StopExe,
    Deceleration := GVL_AXIS4.stWM_VelCmd.lrDeceleration,
    Jerk := GVL_AXIS4.stWM_VelCmd.lrJerk,
    Options := GVL_AXIS4.stWM_VelCmd.EnuOptions,
    Busy => GVL_AXIS4.stWM_Stop.Busy,
    Active => GVL_AXIS4.stWM_Stop.Active,
    CommandAborted => GVL_AXIS4.stWM_Stop.CmdAborted,
    Error => GVL_AXIS4.stWM_Stop.Error,
    ErrorID => GVL_AXIS4.stWM_Stop.ErrorID); // MC_Stop
GVL_AXIS4.stWM_Stop.Done := GVL_AXIS4.fbWM_Stop.Done;

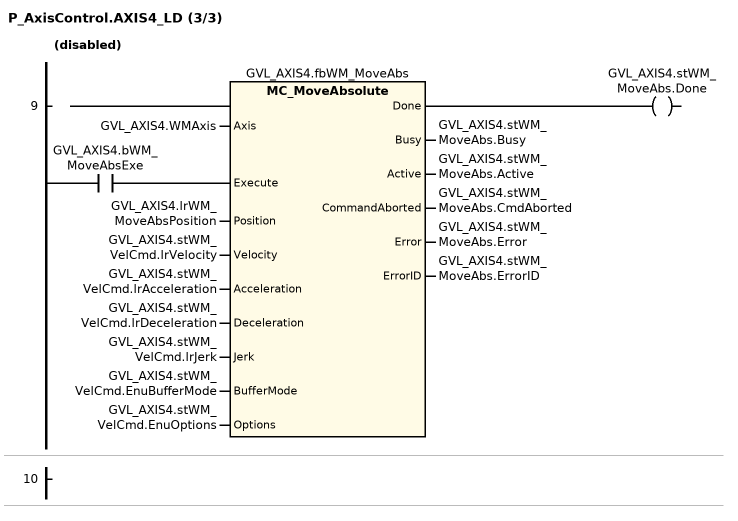
// NETWORK 9 (disabled)
// GVL_AXIS4.fbWM_MoveAbs(
//     Axis := GVL_AXIS4.WMAxis,
//     Execute := GVL_AXIS4.bWM_MoveAbsExe,
//     Position := GVL_AXIS4.lrWM_MoveAbsPosition,
//     Velocity := GVL_AXIS4.stWM_VelCmd.lrVelocity,
//     Acceleration := GVL_AXIS4.stWM_VelCmd.lrAcceleration,
//     Deceleration := GVL_AXIS4.stWM_VelCmd.lrDeceleration,
//     Jerk := GVL_AXIS4.stWM_VelCmd.lrJerk,
//     BufferMode := GVL_AXIS4.stWM_VelCmd.EnuBufferMode,
//     Options := GVL_AXIS4.stWM_VelCmd.EnuOptions,
//     Busy => GVL_AXIS4.stWM_MoveAbs.Busy,
//     Active => GVL_AXIS4.stWM_MoveAbs.Active,
//     CommandAborted => GVL_AXIS4.stWM_MoveAbs.CmdAborted,
//     Error => GVL_AXIS4.stWM_MoveAbs.Error,
//     ErrorID => GVL_AXIS4.stWM_MoveAbs.ErrorID); // MC_MoveAbsolute
// GVL_AXIS4.stWM_MoveAbs.Done := GVL_AXIS4.fbWM_MoveAbs.Done;

// NETWORK 10
END_METHOD

METHOD AXIS4_LD_Auto : BOOL
VAR_INPUT
END_VAR
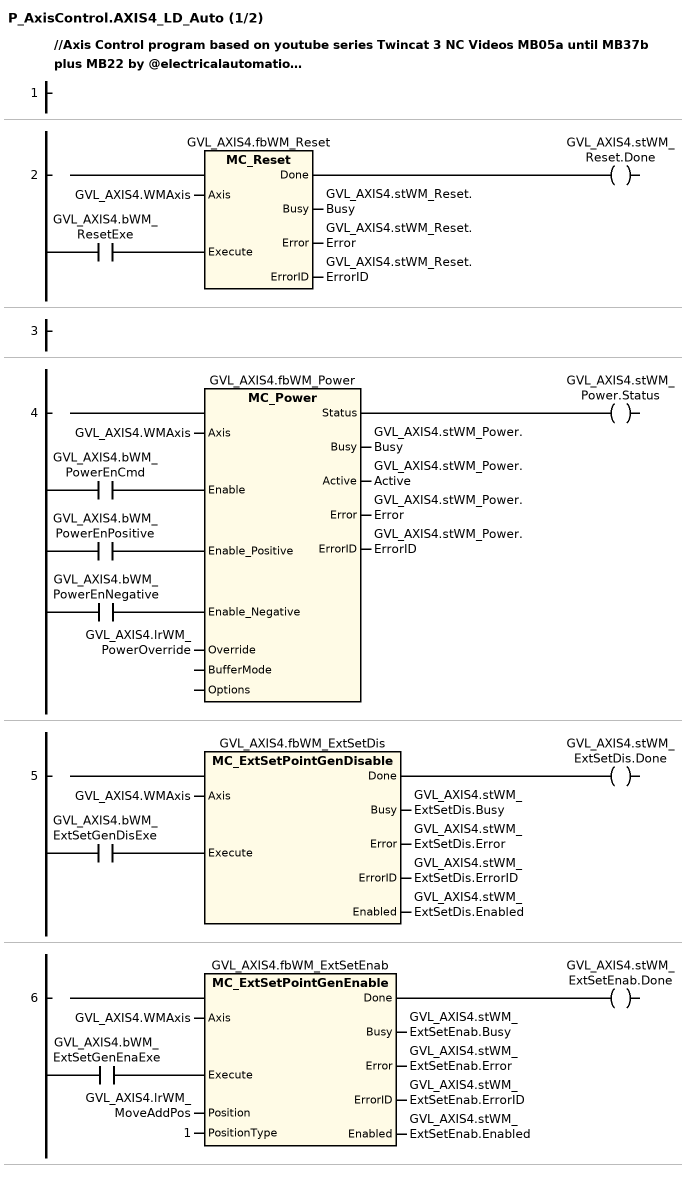
// NETWORK 1: //Axis Control program based on youtube series Twincat 3 NC Videos MB05a until MB37b plus MB22 by @electricalautomation https://www.youtube.com/waWMh?v=BxRAOdTks9I&list=PL762SfoJC-e8NbAUQ-H7a_TOdqrlBPCw4&index=25

// NETWORK 2
GVL_AXIS4.fbWM_Reset(
    Axis := GVL_AXIS4.WMAxis,
    Execute := GVL_AXIS4.bWM_ResetExe,
    Busy => GVL_AXIS4.stWM_Reset.Busy,
    Error => GVL_AXIS4.stWM_Reset.Error,
    ErrorID => GVL_AXIS4.stWM_Reset.ErrorID); // MC_Reset
GVL_AXIS4.stWM_Reset.Done := GVL_AXIS4.fbWM_Reset.Done;

// NETWORK 3

// NETWORK 4
GVL_AXIS4.fbWM_Power(
    Axis := GVL_AXIS4.WMAxis,
    Enable := GVL_AXIS4.bWM_PowerEnCmd,
    Enable_Positive := GVL_AXIS4.bWM_PowerEnPositive,
    Enable_Negative := GVL_AXIS4.bWM_PowerEnNegative,
    Override := GVL_AXIS4.lrWM_PowerOverride,
    Busy => GVL_AXIS4.stWM_Power.Busy,
    Active => GVL_AXIS4.stWM_Power.Active,
    Error => GVL_AXIS4.stWM_Power.Error,
    ErrorID => GVL_AXIS4.stWM_Power.ErrorID); // MC_Power
GVL_AXIS4.stWM_Power.Status := GVL_AXIS4.fbWM_Power.Status;

// NETWORK 5
GVL_AXIS4.fbWM_ExtSetDis(
    Axis := GVL_AXIS4.WMAxis,
    Execute := GVL_AXIS4.bWM_ExtSetGenDisExe,
    Busy => GVL_AXIS4.stWM_ExtSetDis.Busy,
    Error => GVL_AXIS4.stWM_ExtSetDis.Error,
    ErrorID => GVL_AXIS4.stWM_ExtSetDis.ErrorID,
    Enabled => GVL_AXIS4.stWM_ExtSetDis.Enabled); // MC_ExtSetPointGenDisable
GVL_AXIS4.stWM_ExtSetDis.Done := GVL_AXIS4.fbWM_ExtSetDis.Done;

// NETWORK 6
GVL_AXIS4.fbWM_ExtSetEnab(
    Axis := GVL_AXIS4.WMAxis,
    Execute := GVL_AXIS4.bWM_ExtSetGenEnaExe,
    Position := GVL_AXIS4.lrWM_MoveAddPos,
    PositionType := 1,
    Busy => GVL_AXIS4.stWM_ExtSetEnab.Busy,
    Error => GVL_AXIS4.stWM_ExtSetEnab.Error,
    ErrorID => GVL_AXIS4.stWM_ExtSetEnab.ErrorID,
    Enabled => GVL_AXIS4.stWM_ExtSetEnab.Enabled); // MC_ExtSetPointGenEnable
GVL_AXIS4.stWM_ExtSetEnab.Done := GVL_AXIS4.fbWM_ExtSetEnab.Done;

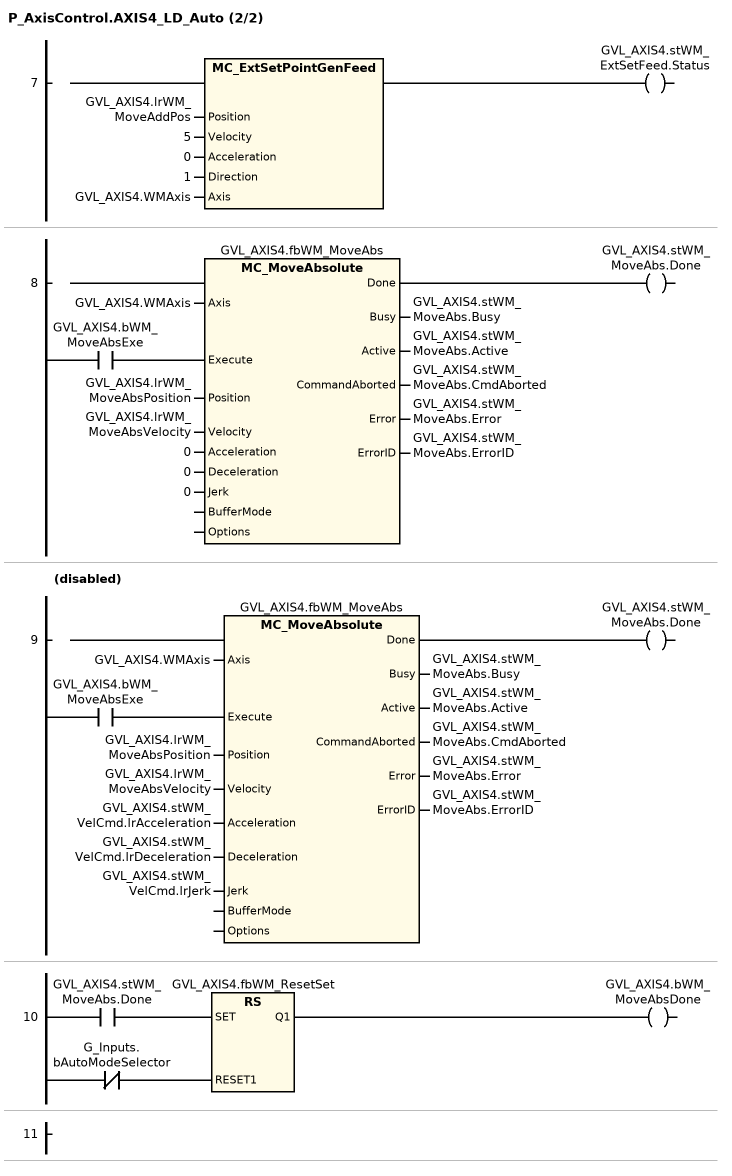
// NETWORK 7
GVL_AXIS4.stWM_ExtSetFeed.Status := MC_ExtSetPointGenFeed(Position := GVL_AXIS4.lrWM_MoveAddPos, Velocity := 5, Acceleration := 0, Direction := 1, Axis := GVL_AXIS4.WMAxis);

// NETWORK 8
GVL_AXIS4.fbWM_MoveAbs(
    Axis := GVL_AXIS4.WMAxis,
    Execute := GVL_AXIS4.bWM_MoveAbsExe,
    Position := GVL_AXIS4.lrWM_MoveAbsPosition,
    Velocity := GVL_AXIS4.lrWM_MoveAbsVelocity,
    Acceleration := 0,
    Deceleration := 0,
    Jerk := 0,
    Busy => GVL_AXIS4.stWM_MoveAbs.Busy,
    Active => GVL_AXIS4.stWM_MoveAbs.Active,
    CommandAborted => GVL_AXIS4.stWM_MoveAbs.CmdAborted,
    Error => GVL_AXIS4.stWM_MoveAbs.Error,
    ErrorID => GVL_AXIS4.stWM_MoveAbs.ErrorID); // MC_MoveAbsolute
GVL_AXIS4.stWM_MoveAbs.Done := GVL_AXIS4.fbWM_MoveAbs.Done;

// NETWORK 9 (disabled)
// GVL_AXIS4.fbWM_MoveAbs(
//     Axis := GVL_AXIS4.WMAxis,
//     Execute := GVL_AXIS4.bWM_MoveAbsExe,
//     Position := GVL_AXIS4.lrWM_MoveAbsPosition,
//     Velocity := GVL_AXIS4.lrWM_MoveAbsVelocity,
//     Acceleration := GVL_AXIS4.stWM_VelCmd.lrAcceleration,
//     Deceleration := GVL_AXIS4.stWM_VelCmd.lrDeceleration,
//     Jerk := GVL_AXIS4.stWM_VelCmd.lrJerk,
//     Busy => GVL_AXIS4.stWM_MoveAbs.Busy,
//     Active => GVL_AXIS4.stWM_MoveAbs.Active,
//     CommandAborted => GVL_AXIS4.stWM_MoveAbs.CmdAborted,
//     Error => GVL_AXIS4.stWM_MoveAbs.Error,
//     ErrorID => GVL_AXIS4.stWM_MoveAbs.ErrorID); // MC_MoveAbsolute
// GVL_AXIS4.stWM_MoveAbs.Done := GVL_AXIS4.fbWM_MoveAbs.Done;

// NETWORK 10
GVL_AXIS4.fbWM_ResetSet(SET := GVL_AXIS4.stWM_MoveAbs.Done, RESET1 := NOT G_Inputs.bAutoModeSelector); // RS
GVL_AXIS4.bWM_MoveAbsDone := GVL_AXIS4.fbWM_ResetSet.Q1;

// NETWORK 11
END_METHOD

METHOD Manual_mode : BOOL
VAR_INPUT
END_VAR
//Axis 1 Main arm actuator
AXIS1_LD();

GVL_AXIS1.bBC_ResetExe := FALSE;

GVL_AXIS1.stBC_VelCmd.EnuDirection := MC_Undefined_Direction;

GVL_AXIS1.stBC_VelCmd.bExe := FALSE;

GVL_AXIS1.bBC_PowerEnCmd := G_Inputs.bManualModeSelector;

IF G_Sensors.fJoystickLeftNormalizedX  > 0 AND G_Inputs.bJoystickLeftEnable THEN
	GVL_AXIS1.bBC_PowerEnNegative := TRUE;
	GVL_AXIS1.stBC_VelCmd.EnuDirection := MC_Negative_Direction;
	GVL_AXIS1.lrBC_PowerOverride := ABS(G_Sensors.fJoystickLeftNormalizedX) * 100;	
	GVL_AXIS1.stBC_VelCmd.bExe := TRUE;
ELSIF G_Sensors.fJoystickLeftNormalizedX < 0 AND G_Inputs.bJoystickLeftEnable THEN
	GVL_AXIS1.bBC_PowerEnPositive := TRUE;
	GVL_AXIS1.stBC_VelCmd.EnuDirection := MC_Positive_Direction;
	GVL_AXIS1.lrBC_PowerOverride := ABS(G_Sensors.fJoystickLeftNormalizedX) * 100;	
	GVL_AXIS1.stBC_VelCmd.bExe := TRUE;
ELSE
	 GVL_AXIS1.lrBC_PowerOverride := 0;
	 GVL_AXIS1.stBC_VelCmd.bExe := FALSE;
	 GVL_AXIS1.bBC_PowerEnNegative := FALSE;
	 GVL_AXIS1.bBC_PowerEnPositive := FALSE;
END_IF

GVL_AXIS1.bBC_ResetExe := TRUE;


//Axis 2 Slew joint actuator
AXIS2_LD();

GVL_AXIS2.bSJ_ResetExe := FALSE;

GVL_AXIS2.stSJ_VelCmd.EnuDirection := MC_Undefined_Direction;

GVL_AXIS2.stSJ_VelCmd.bExe := FALSE;

GVL_AXIS2.bSJ_PowerEnCmd := G_Inputs.bManualModeSelector;

IF G_Sensors.fJoystickRightNormalizedX  > 0 AND G_Inputs.bJoystickRightEnable THEN
	GVL_AXIS2.bSJ_PowerEnPositive := TRUE;
	GVL_AXIS2.stSJ_VelCmd.EnuDirection := MC_Positive_Direction;
	GVL_AXIS2.lrSJ_PowerOverride := ABS(G_Sensors.fJoystickRightNormalizedX) * 100;	
	GVL_AXIS2.stSJ_VelCmd.bExe := TRUE;
ELSIF G_Sensors.fJoystickRightNormalizedX < 0 AND G_Inputs.bJoystickRightEnable THEN
	GVL_AXIS2.bSJ_PowerEnNegative := TRUE;
	GVL_AXIS2.stSJ_VelCmd.EnuDirection := MC_Negative_Direction;
	GVL_AXIS2.lrSJ_PowerOverride := ABS(G_Sensors.fJoystickRightNormalizedX) * 100;	
	GVL_AXIS2.stSJ_VelCmd.bExe := TRUE;
ELSE
	 GVL_AXIS2.lrSJ_PowerOverride := 0;
	 GVL_AXIS2.stSJ_VelCmd.bExe := FALSE;
	 GVL_AXIS2.bSJ_PowerEnNegative := FALSE;
	 GVL_AXIS2.bSJ_PowerEnPositive := FALSE;
END_IF

GVL_AXIS2.bSJ_ResetExe := TRUE;


//Axis 3 Knuckle arm actuator
AXIS3_LD();

GVL_AXIS3.bTC_ResetExe := FALSE;

GVL_AXIS3.stTC_VelCmd.EnuDirection := MC_Undefined_Direction;

GVL_AXIS3.stTC_VelCmd.bExe := FALSE;

GVL_AXIS3.bTC_PowerEnCmd := G_Inputs.bManualModeSelector;

IF G_Sensors.fJoystickLeftNormalizedY  > 0 AND G_Inputs.bJoystickLeftEnable THEN
	GVL_AXIS3.bTC_PowerEnPositive := TRUE;
	GVL_AXIS3.stTC_VelCmd.EnuDirection := MC_Positive_Direction;
	GVL_AXIS3.lrTC_PowerOverride := ABS(G_Sensors.fJoystickLeftNormalizedY) * 100;	
	GVL_AXIS3.stTC_VelCmd.bExe := TRUE;
ELSIF G_Sensors.fJoystickLeftNormalizedY < 0 AND G_Inputs.bJoystickLeftEnable THEN
	GVL_AXIS3.bTC_PowerEnNegative := TRUE;
	GVL_AXIS3.stTC_VelCmd.EnuDirection := MC_Negative_Direction;
	GVL_AXIS3.lrTC_PowerOverride := ABS(G_Sensors.fJoystickLeftNormalizedY) * 100;	
	GVL_AXIS3.stTC_VelCmd.bExe := TRUE;
ELSE
	 GVL_AXIS3.lrTC_PowerOverride := 0;
	 GVL_AXIS3.stTC_VelCmd.bExe := FALSE;
	 GVL_AXIS3.bTC_PowerEnNegative := FALSE;
	 GVL_AXIS3.bTC_PowerEnPositive := FALSE;
END_IF

GVL_AXIS3.bTC_ResetExe := TRUE;

(*
AXIS3_LD();

GVL_AXIS3.bTC_ResetExe := G_Inputs.bJoystickLeftEnable;

GVL_AXIS3.EnuMoveVelDirection := G_Sensors.MCDirectionAxis3;

GVL_AXIS3.bTC_PowerEnCmd := G_Inputs.bManualModeSelector;
GVL_AXIS3.bTC_PowerEnNegative := G_Inputs.bManualModeSelector;
GVL_AXIS3.bTC_PowerEnPositive := G_Inputs.bManualModeSelector;


// Velocity control
IF G_Sensors.fJoystickLeftNormalizedY  > 0.01 AND G_Inputs.bJoystickLeftEnable THEN
	GVL_AXIS3.stTC_VelCmd.EnuDirection := MC_Positive_Direction;
	GVL_AXIS3.lrTC_PowerOverride := ABS(G_Sensors.fJoystickLeftNormalizedY) * 100;	
	GVL_AXIS3.stTC_VelCmd.bExe := TRUE;
ELSIF G_Sensors.fJoystickLeftNormalizedY < 0.01 AND G_Inputs.bJoystickLeftEnable THEN
	GVL_AXIS3.stTC_VelCmd.EnuDirection := MC_Negative_Direction;
	GVL_AXIS3.lrTC_PowerOverride := ABS(G_Sensors.fJoystickLeftNormalizedY) * 100;	
	GVL_AXIS3.stTC_VelCmd.bExe := TRUE;
ELSE
	 GVL_AXIS3.lrTC_PowerOverride := 0;
	 //GVL_AXIS3.stTC_VelCmd.EnuDirection := MC_Current_Direction;
	 GVL_AXIS3.stTC_VelCmd.bExe := FALSE;
END_IF
*)

(*
AXIS4_LD();

GVL_AXIS4.bWM_ResetExe := G_Inputs.bJoystickRightEnable;

GVL_AXIS4.EnuMoveVelDirection := G_Sensors.MCDirectionAxis4;

GVL_AXIS4.bWM_PowerEnCmd := G_Inputs.bManualModeSelector;
GVL_AXIS4.bWM_PowerEnNegative := G_Inputs.bManualModeSelector;
GVL_AXIS4.bWM_PowerEnPositive := G_Inputs.bManualModeSelector;


// Velocity control
IF G_Sensors.fJoystickLeftNormalizedY  > 0 AND G_Inputs.bJoystickRightEnable THEN
	GVL_AXIS4.lrWM_PowerOverride := ABS(G_Sensors.fJoystickRightNormalizedY) * 100;
	GVL_AXIS4.stWM_VelCmd.EnuDirection := MC_Positive_Direction;
	GVL_AXIS4.stWM_VelCmd.bExe := TRUE;
ELSIF G_Sensors.fJoystickLeftNormalizedY < 0 AND G_Inputs.bJoystickLeftEnable THEN
	GVL_AXIS4.lrWM_PowerOverride := ABS(G_Sensors.fJoystickLeftNormalizedY) * 100;
	GVL_AXIS4.stWM_VelCmd.EnuDirection := MC_Negative_Direction;
	GVL_AXIS4.stWM_VelCmd.bExe := TRUE;
ELSE
	 GVL_AXIS4.lrWM_PowerOverride := 0;
	 GVL_AXIS4.stWM_VelCmd.EnuDirection := MC_Current_Direction;
	 GVL_AXIS4.stWM_VelCmd.bExe := FALSE;
END_IF
*)

//Axis 4 Winch motor actuator
AXIS4_LD();

GVL_AXIS4.bWM_ResetExe := FALSE;

GVL_AXIS4.stWM_VelCmd.EnuDirection := MC_Undefined_Direction;

GVL_AXIS4.stWM_VelCmd.bExe := FALSE;

GVL_AXIS4.bWM_PowerEnCmd := G_Inputs.bManualModeSelector;

IF G_Sensors.fJoystickRightNormalizedY  > 0 AND G_Inputs.bJoystickRightEnable THEN
	GVL_AXIS4.bWM_PowerEnNegative := TRUE;
	GVL_AXIS4.stWM_VelCmd.EnuDirection := MC_Negative_Direction;
	GVL_AXIS4.lrWM_PowerOverride := ABS(G_Sensors.fJoystickRightNormalizedY) * 100;	
	GVL_AXIS4.stWM_VelCmd.bExe := TRUE;
ELSIF G_Sensors.fJoystickRightNormalizedY < 0 AND G_Inputs.bJoystickRightEnable THEN
	GVL_AXIS4.bWM_PowerEnPositive := TRUE;
	GVL_AXIS4.stWM_VelCmd.EnuDirection := MC_Positive_Direction;
	GVL_AXIS4.lrWM_PowerOverride := ABS(G_Sensors.fJoystickRightNormalizedY) * 100;	
	GVL_AXIS4.stWM_VelCmd.bExe := TRUE;
ELSE
	 GVL_AXIS4.lrWM_PowerOverride := 0;
	 GVL_AXIS4.stWM_VelCmd.bExe := FALSE;
	 GVL_AXIS4.bWM_PowerEnNegative := FALSE;
	 GVL_AXIS4.bWM_PowerEnPositive := FALSE;
END_IF

GVL_AXIS4.bWM_ResetExe := TRUE;
END_METHOD

END_PROGRAM

(* stored: Version 1.1.0.1, ProductVersion 3.1.4024.12
   POU P_AxisControl: Id {5037aaa5-6389-4d48-9944-f1b3147b0b82}, SpecialFunc None
   Method Auto_mode: Id {d04e60f4-7a42-4fb1-907e-93e16dbafa43}
   Method AXIS1_LD: Id {a2ea73c2-d9a7-46bb-9d54-a37d5bff0a65}
   Method AXIS1_LD_Auto: Id {30907942-6a1d-4345-9aab-8829bd87d527}
   Method AXIS2_LD: Id {bdec519a-41ff-484d-9600-76653e24e62b}
   Method AXIS3_LD: Id {3773e93e-9c66-4353-b78a-0a74486d73ef}
   Method AXIS3_LD_Auto: Id {0b7586c2-7587-4f9c-ad47-7bf16864663e}
   Method AXIS4_LD: Id {c68d9161-8577-4188-91d1-8d05a7c19713}
   Method AXIS4_LD_Auto: Id {8b81b91c-b043-4745-82a0-5697b09e72c1}
   Method Manual_mode: Id {1fd68a25-3da3-4bba-af59-1b4dc6fc6de5} *)
